FUNCTION_BLOCK Section2
  (* Standard: 61499-2 *)
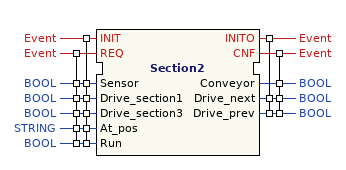
  EVENT_INPUT
    INIT WITH Sensor, Drive_section1, Drive_section3, At_pos, Run;
    REQ WITH Sensor, Drive_section1, Drive_section3, At_pos, Run;
  END_EVENT
  EVENT_OUTPUT
    INITO WITH Drive_next, Drive_prev;
    CNF WITH Drive_next, Drive_prev, Conveyor;
  END_EVENT
  VAR_INPUT
    Sensor : BOOL;
    Drive_section1 : BOOL;
    Drive_section3 : BOOL;
    At_pos : STRING;
    Run : BOOL;
  END_VAR
  VAR_OUTPUT
    Conveyor : BOOL;
    Drive_next : BOOL;
    Drive_prev : BOOL;
  END_VAR
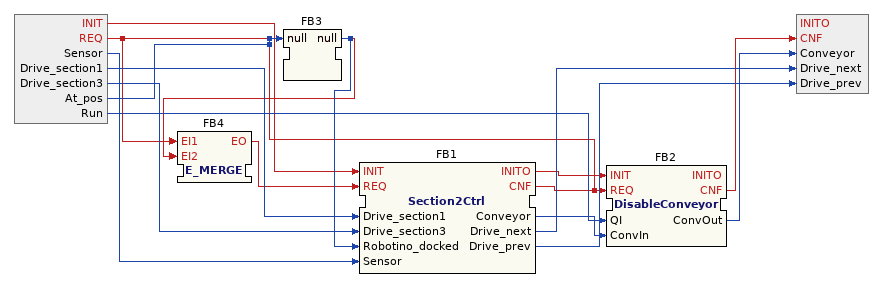
  FBS
    FB1 : Section2Ctrl;
    FB2 : DisableConveyor;
    FB3 : ;
    FB4 : E_MERGE;
  END_FBS
  EVENT_CONNECTIONS
    REQ TO FB4.EI1;
    FB1.INITO TO FB2.INIT;
    INIT TO FB1.INIT;
    FB1.CNF TO FB2.REQ;
    REQ TO FB2.REQ;
    FB2.CNF TO CNF;
    FB3.null TO FB4.EI2;
    FB4.EO TO FB1.REQ;
    REQ TO FB3.null;
  END_CONNECTIONS
  DATA_CONNECTIONS
    Drive_section1 TO FB1.Drive_section1;
    Drive_section3 TO FB1.Drive_section3;
    FB1.Drive_next TO Drive_next;
    FB1.Drive_prev TO Drive_prev;
    FB1.Conveyor TO FB2.ConvIn;
    Run TO FB2.QI;
    FB2.ConvOut TO Conveyor;
    Sensor TO FB1.Sensor;
    At_pos TO FB3.null;
    FB3.null TO FB1.Robotino_docked;
  END_CONNECTIONS
END_FUNCTION_BLOCK
